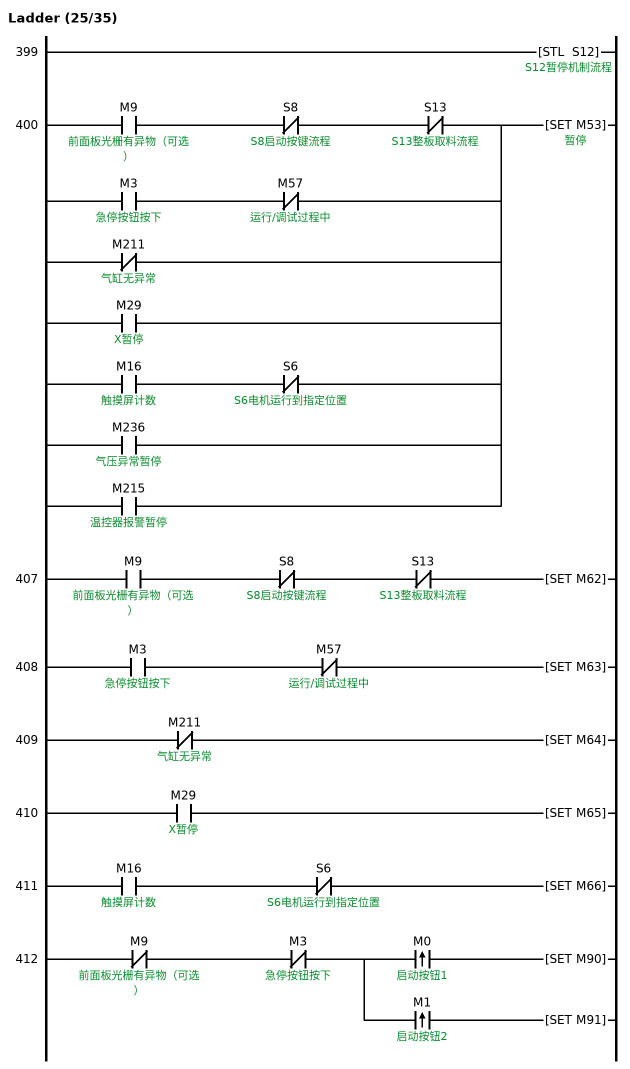
[picture p24: Ladder rows 399-412]
STL    S12	; S12暂停机制流程
LD     M9	; 前面板光栅有异物（可选）
ANI    S8	; S8启动按键流程
ANI    S13	; S13整板取料流程
LD     M3	; 急停按钮按下
ANI    M57	; 运行/调试过程中
ORB
ORI    M211	; 气缸无异常
OR     M29	; X暂停
LD     M16	; 触摸屏计数
ANI    S6	; S6电机运行到指定位置
ORB
OR     M236	; 气压异常暂停
OR     M215	; 温控器报警暂停
SET    M53	; 暂停
LD     M9	; 前面板光栅有异物（可选）
ANI    S8	; S8启动按键流程
ANI    S13	; S13整板取料流程
SET    M62
LD     M3	; 急停按钮按下
ANI    M57	; 运行/调试过程中
SET    M63
LDI    M211	; 气缸无异常
SET    M64
LD     M29	; X暂停
SET    M65
LD     M16	; 触摸屏计数
ANI    S6	; S6电机运行到指定位置
SET    M66
LDI    M9	; 前面板光栅有异物（可选）
ANI    M3	; 急停按钮按下
MPS
ANDP   M0	; 启动按钮1
SET    M90
MPP
ANDP   M1	; 启动按钮2
SET    M91

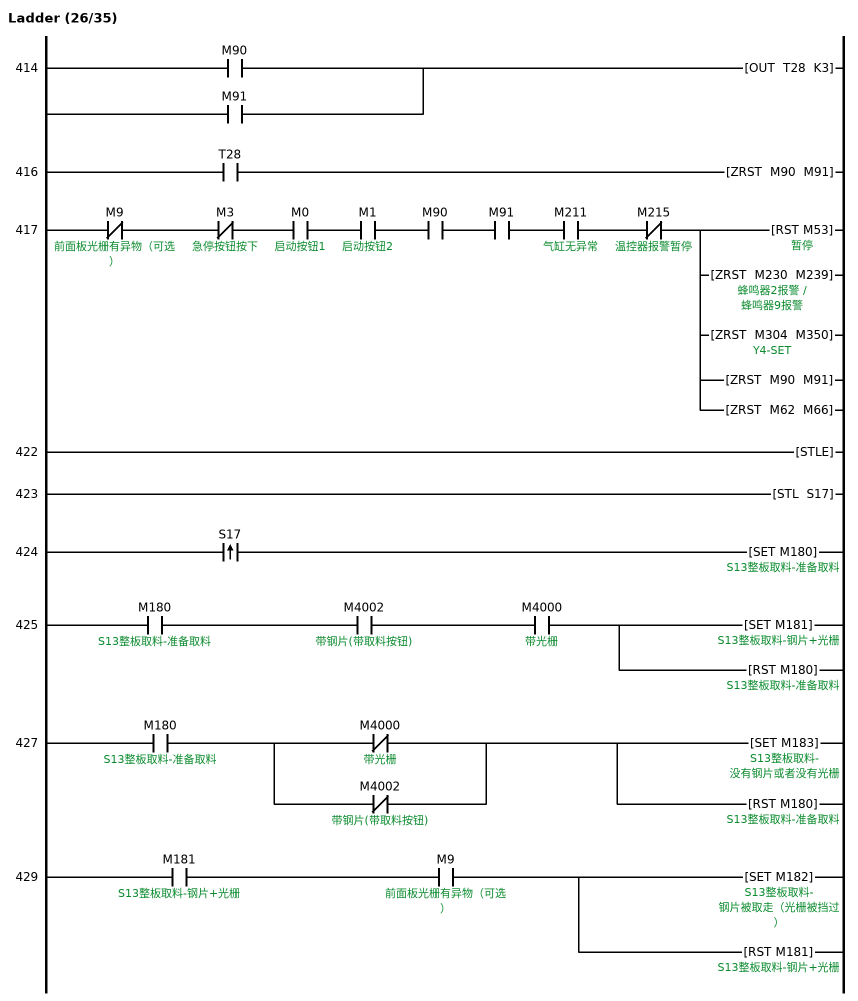
LD     M90
OR     M91
OUT    T28 K3
LD     T28
ZRST   M90 M91
LDI    M9	; 前面板光栅有异物（可选）
ANI    M3	; 急停按钮按下
AND    M0	; 启动按钮1
AND    M1	; 启动按钮2
AND    M90
AND    M91
AND    M211	; 气缸无异常
ANI    M215	; 温控器报警暂停
RST    M53	; 暂停
ZRST   M230 M239	; 蜂鸣器2报警 / 蜂鸣器9报警
ZRST   M304 M350	; Y4-SET
ZRST   M90 M91
ZRST   M62 M66
STLE
STL    S17
LDP    S17
SET    M180	; S13整板取料-准备取料
LD     M180	; S13整板取料-准备取料
AND    M4002	; 带钢片(带取料按钮)
AND    M4000	; 带光栅
SET    M181	; S13整板取料-钢片+光栅
RST    M180	; S13整板取料-准备取料
LD     M180	; S13整板取料-准备取料
LDI    M4000	; 带光栅
ORI    M4002	; 带钢片(带取料按钮)
ANB
SET    M183	; S13整板取料-没有钢片或者没有光栅
RST    M180	; S13整板取料-准备取料
LD     M181	; S13整板取料-钢片+光栅
AND    M9	; 前面板光栅有异物（可选）
SET    M182	; S13整板取料-钢片被取走（光栅被挡过）
RST    M181	; S13整板取料-钢片+光栅

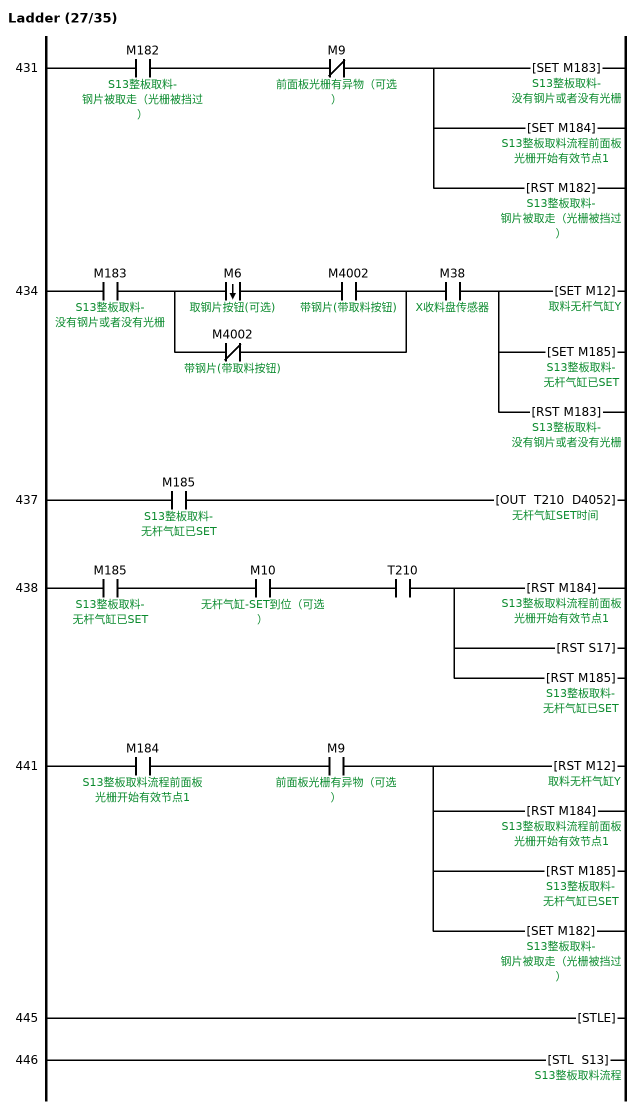
LD     M182	; S13整板取料-钢片被取走（光栅被挡过）
ANI    M9	; 前面板光栅有异物（可选）
SET    M183	; S13整板取料-没有钢片或者没有光栅
SET    M184	; S13整板取料流程前面板光栅开始有效节点1
RST    M182	; S13整板取料-钢片被取走（光栅被挡过）
LD     M183	; S13整板取料-没有钢片或者没有光栅
LDF    M6	; 取钢片按钮(可选)
AND    M4002	; 带钢片(带取料按钮)
ORI    M4002	; 带钢片(带取料按钮)
ANB
AND    M38	; X收料盘传感器
SET    M12	; 取料无杆气缸Y
SET    M185	; S13整板取料-无杆气缸已SET
RST    M183	; S13整板取料-没有钢片或者没有光栅
LD     M185	; S13整板取料-无杆气缸已SET
OUT    T210 D4052	; 无杆气缸SET时间
LD     M185	; S13整板取料-无杆气缸已SET
AND    M10	; 无杆气缸-SET到位（可选）
AND    T210
RST    M184	; S13整板取料流程前面板光栅开始有效节点1
RST    S17
RST    M185	; S13整板取料-无杆气缸已SET
LD     M184	; S13整板取料流程前面板光栅开始有效节点1
AND    M9	; 前面板光栅有异物（可选）
RST    M12	; 取料无杆气缸Y
RST    M184	; S13整板取料流程前面板光栅开始有效节点1
RST    M185	; S13整板取料-无杆气缸已SET
SET    M182	; S13整板取料-钢片被取走（光栅被挡过）
STLE
STL    S13	; S13整板取料流程

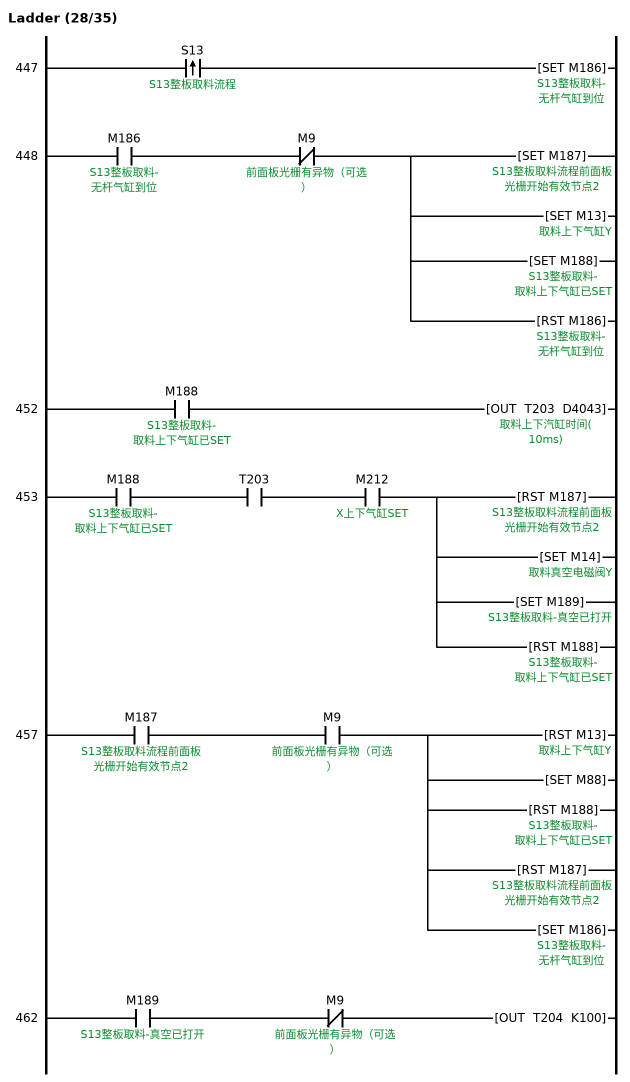
LDP    S13	; S13整板取料流程
SET    M186	; S13整板取料-无杆气缸到位
LD     M186	; S13整板取料-无杆气缸到位
ANI    M9	; 前面板光栅有异物（可选）
SET    M187	; S13整板取料流程前面板光栅开始有效节点2
SET    M13	; 取料上下气缸Y
SET    M188	; S13整板取料-取料上下气缸已SET
RST    M186	; S13整板取料-无杆气缸到位
LD     M188	; S13整板取料-取料上下气缸已SET
OUT    T203 D4043	; 取料上下汽缸时间(10ms)
LD     M188	; S13整板取料-取料上下气缸已SET
AND    T203
AND    M212	; X上下气缸SET
RST    M187	; S13整板取料流程前面板光栅开始有效节点2
SET    M14	; 取料真空电磁阀Y
SET    M189	; S13整板取料-真空已打开
RST    M188	; S13整板取料-取料上下气缸已SET
LD     M187	; S13整板取料流程前面板光栅开始有效节点2
AND    M9	; 前面板光栅有异物（可选）
RST    M13	; 取料上下气缸Y
SET    M88
RST    M188	; S13整板取料-取料上下气缸已SET
RST    M187	; S13整板取料流程前面板光栅开始有效节点2
SET    M186	; S13整板取料-无杆气缸到位
LD     M189	; S13整板取料-真空已打开
ANI    M9	; 前面板光栅有异物（可选）
OUT    T204 K100

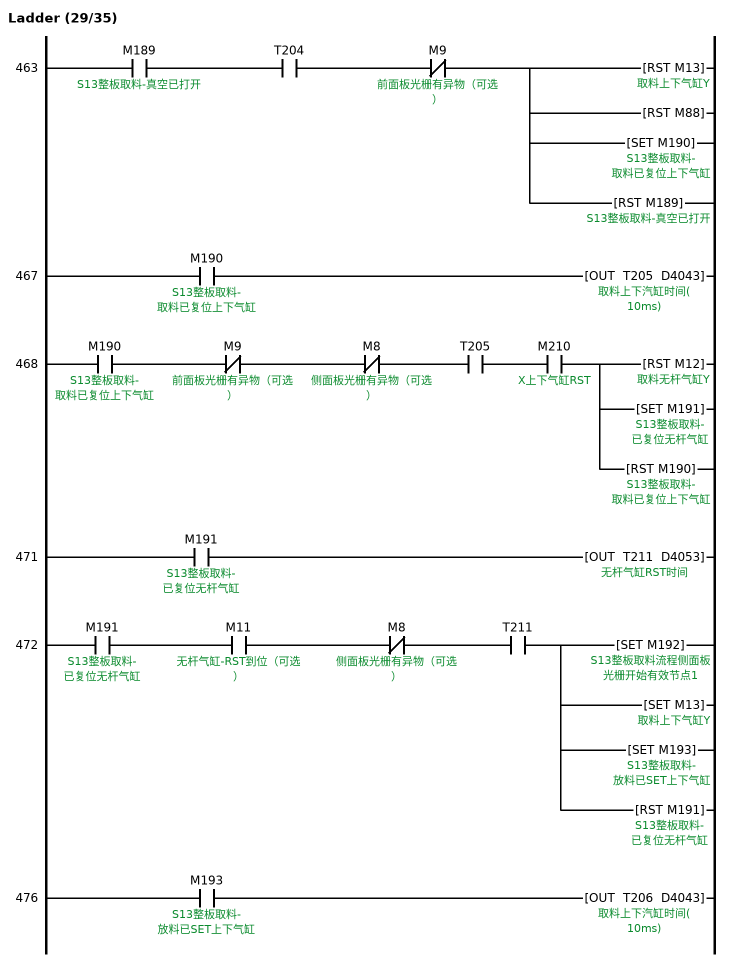
LD     M189	; S13整板取料-真空已打开
AND    T204
ANI    M9	; 前面板光栅有异物（可选）
RST    M13	; 取料上下气缸Y
RST    M88
SET    M190	; S13整板取料-取料已复位上下气缸
RST    M189	; S13整板取料-真空已打开
LD     M190	; S13整板取料-取料已复位上下气缸
OUT    T205 D4043	; 取料上下汽缸时间(10ms)
LD     M190	; S13整板取料-取料已复位上下气缸
ANI    M9	; 前面板光栅有异物（可选）
ANI    M8	; 侧面板光栅有异物（可选）
AND    T205
AND    M210	; X上下气缸RST
RST    M12	; 取料无杆气缸Y
SET    M191	; S13整板取料-已复位无杆气缸
RST    M190	; S13整板取料-取料已复位上下气缸
LD     M191	; S13整板取料-已复位无杆气缸
OUT    T211 D4053	; 无杆气缸RST时间
LD     M191	; S13整板取料-已复位无杆气缸
AND    M11	; 无杆气缸-RST到位（可选）
ANI    M8	; 侧面板光栅有异物（可选）
AND    T211
SET    M192	; S13整板取料流程侧面板光栅开始有效节点1
SET    M13	; 取料上下气缸Y
SET    M193	; S13整板取料-放料已SET上下气缸
RST    M191	; S13整板取料-已复位无杆气缸
LD     M193	; S13整板取料-放料已SET上下气缸
OUT    T206 D4043	; 取料上下汽缸时间(10ms)

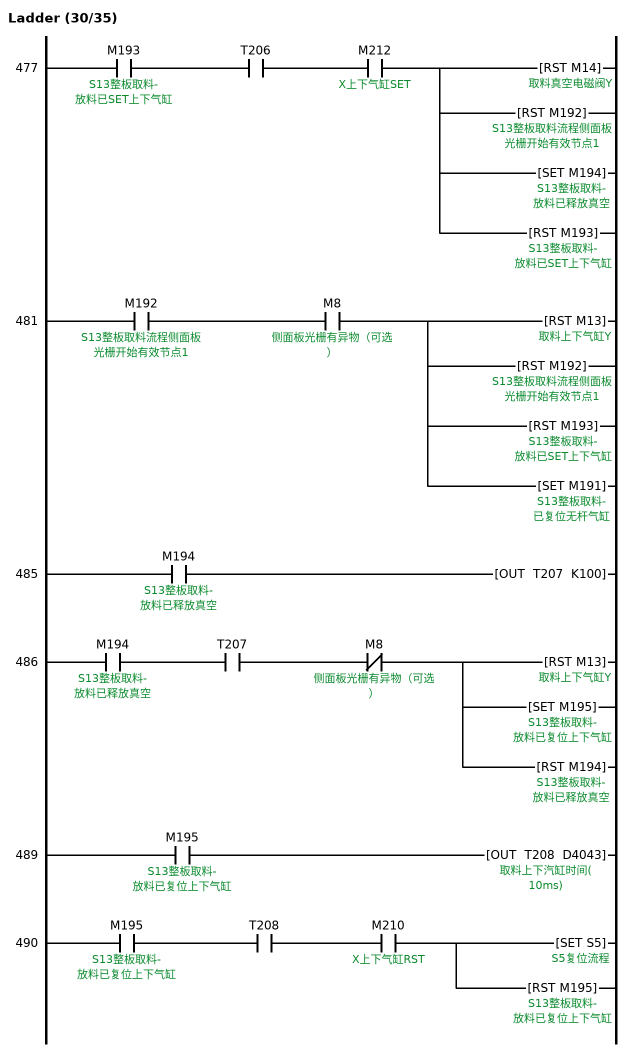
LD     M193	; S13整板取料-放料已SET上下气缸
AND    T206
AND    M212	; X上下气缸SET
RST    M14	; 取料真空电磁阀Y
RST    M192	; S13整板取料流程侧面板光栅开始有效节点1
SET    M194	; S13整板取料-放料已释放真空
RST    M193	; S13整板取料-放料已SET上下气缸
LD     M192	; S13整板取料流程侧面板光栅开始有效节点1
AND    M8	; 侧面板光栅有异物（可选）
RST    M13	; 取料上下气缸Y
RST    M192	; S13整板取料流程侧面板光栅开始有效节点1
RST    M193	; S13整板取料-放料已SET上下气缸
SET    M191	; S13整板取料-已复位无杆气缸
LD     M194	; S13整板取料-放料已释放真空
OUT    T207 K100
LD     M194	; S13整板取料-放料已释放真空
AND    T207
ANI    M8	; 侧面板光栅有异物（可选）
RST    M13	; 取料上下气缸Y
SET    M195	; S13整板取料-放料已复位上下气缸
RST    M194	; S13整板取料-放料已释放真空
LD     M195	; S13整板取料-放料已复位上下气缸
OUT    T208 D4043	; 取料上下汽缸时间(10ms)
LD     M195	; S13整板取料-放料已复位上下气缸
AND    T208
AND    M210	; X上下气缸RST
SET    S5	; S5复位流程
RST    M195	; S13整板取料-放料已复位上下气缸

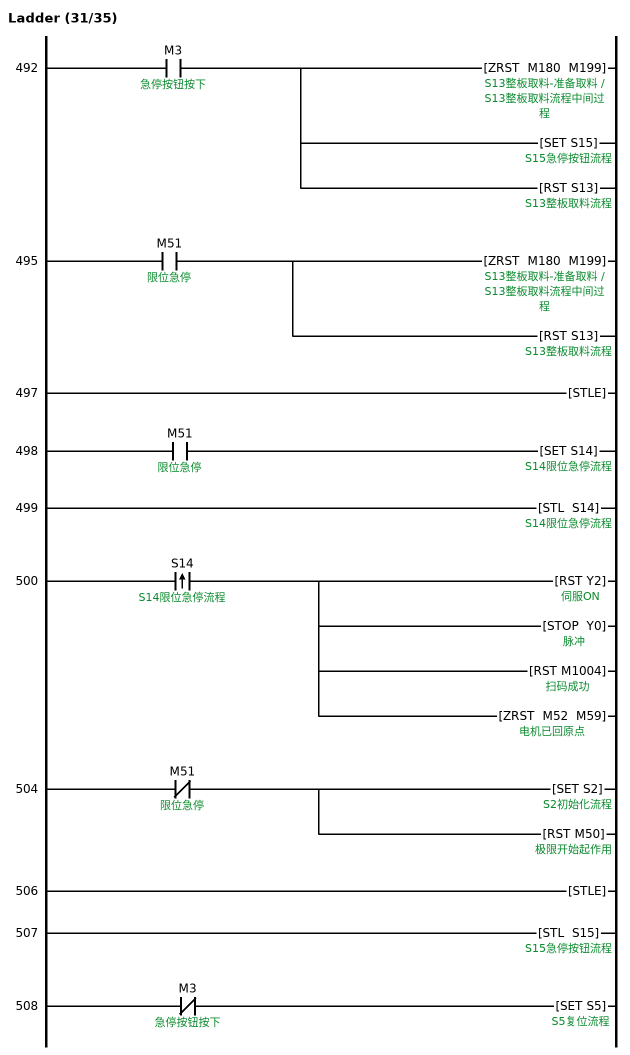
LD     M3	; 急停按钮按下
ZRST   M180 M199	; S13整板取料-准备取料 / S13整板取料流程中间过程
SET    S15	; S15急停按钮流程
RST    S13	; S13整板取料流程
LD     M51	; 限位急停
ZRST   M180 M199	; S13整板取料-准备取料 / S13整板取料流程中间过程
RST    S13	; S13整板取料流程
STLE
LD     M51	; 限位急停
SET    S14	; S14限位急停流程
STL    S14	; S14限位急停流程
LDP    S14	; S14限位急停流程
RST    Y2	; 伺服ON
STOP   Y0	; 脉冲
RST    M1004	; 扫码成功
ZRST   M52 M59	; 电机已回原点
LDI    M51	; 限位急停
SET    S2	; S2初始化流程
RST    M50	; 极限开始起作用
STLE
STL    S15	; S15急停按钮流程
LDI    M3	; 急停按钮按下
SET    S5	; S5复位流程

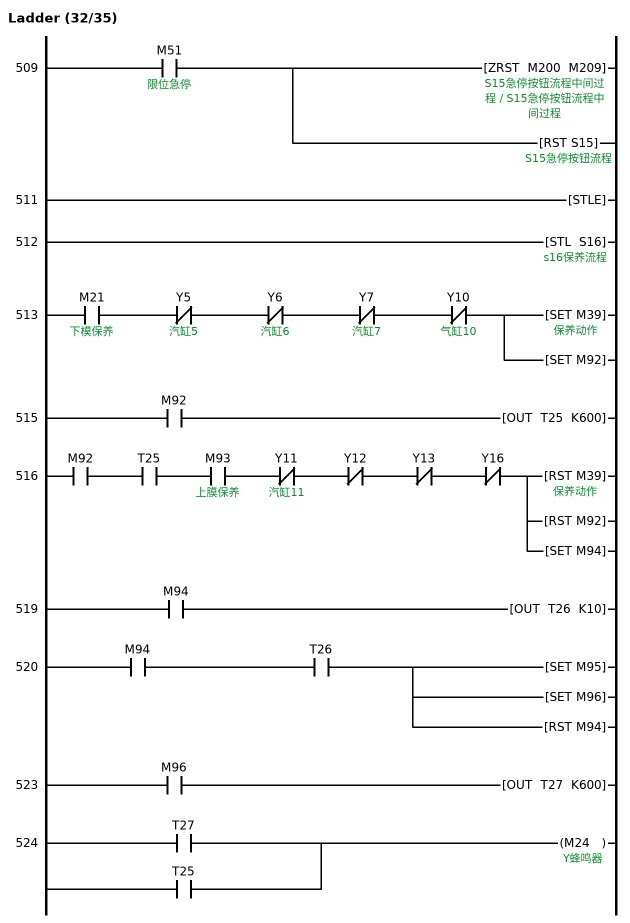
LD     M51	; 限位急停
ZRST   M200 M209	; S15急停按钮流程中间过程 / S15急停按钮流程中间过程
RST    S15	; S15急停按钮流程
STLE
STL    S16	; s16保养流程
LD     M21	; 下模保养
ANI    Y5	; 汽缸5
ANI    Y6	; 汽缸6
ANI    Y7	; 汽缸7
ANI    Y10	; 气缸10
SET    M39	; 保养动作
SET    M92
LD     M92
OUT    T25 K600
LD     M92
AND    T25
AND    M93	; 上膜保养
ANI    Y11	; 汽缸11
ANI    Y12
ANI    Y13
ANI    Y16
RST    M39	; 保养动作
RST    M92
SET    M94
LD     M94
OUT    T26 K10
LD     M94
AND    T26
SET    M95
SET    M96
RST    M94
LD     M96
OUT    T27 K600
LD     T27
OR     T25
OUT    M24	; Y蜂鸣器

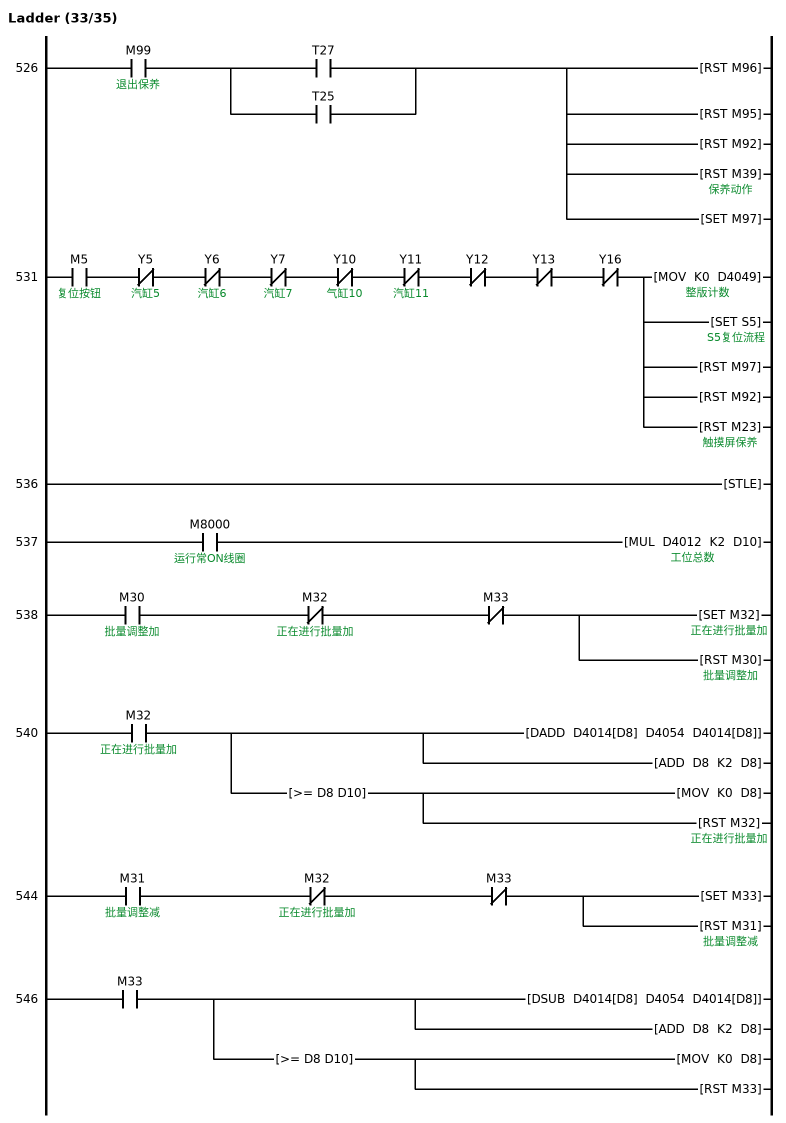
LD     M99	; 退出保养
LD     T27
OR     T25
ANB
RST    M96
RST    M95
RST    M92
RST    M39	; 保养动作
SET    M97
LD     M5	; 复位按钮
ANI    Y5	; 汽缸5
ANI    Y6	; 汽缸6
ANI    Y7	; 汽缸7
ANI    Y10	; 气缸10
ANI    Y11	; 汽缸11
ANI    Y12
ANI    Y13
ANI    Y16
MOV    K0 D4049	; 整版计数
SET    S5	; S5复位流程
RST    M97
RST    M92
RST    M23	; 触摸屏保养
STLE
LD     M8000	; 运行常ON线圈
MUL    D4012 K2 D10	; 工位总数
LD     M30	; 批量调整加
ANI    M32	; 正在进行批量加
ANI    M33
SET    M32	; 正在进行批量加
RST    M30	; 批量调整加
LD     M32	; 正在进行批量加
DADD   D4014[D8] D4054 D4014[D8]
ADD    D8 K2 D8
AND>=  D8 D10
MOV    K0 D8
RST    M32	; 正在进行批量加
LD     M31	; 批量调整减
ANI    M32	; 正在进行批量加
ANI    M33
SET    M33
RST    M31	; 批量调整减
LD     M33
DSUB   D4014[D8] D4054 D4014[D8]
ADD    D8 K2 D8
AND>=  D8 D10
MOV    K0 D8
RST    M33

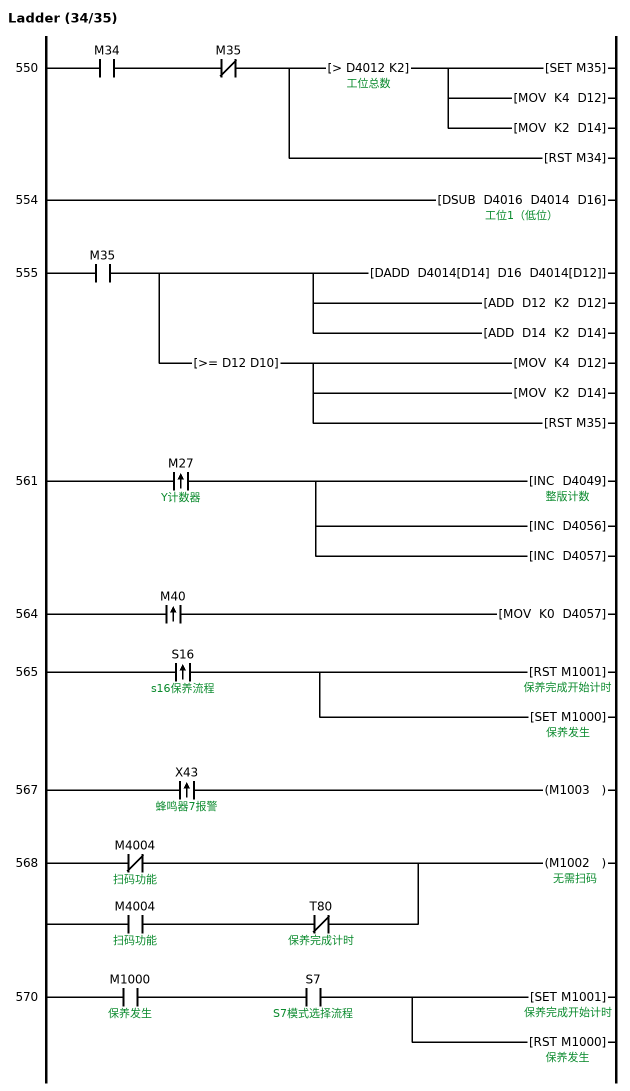
LD     M34
ANI    M35
MPS
AND>   D4012 K2	; 工位总数
SET    M35
MOV    K4 D12
MOV    K2 D14
MPP
RST    M34
DSUB   D4016 D4014 D16	; 工位1（低位）
LD     M35
DADD   D4014[D14] D16 D4014[D12]
ADD    D12 K2 D12
ADD    D14 K2 D14
AND>=  D12 D10
MOV    K4 D12
MOV    K2 D14
RST    M35
LDP    M27	; Y计数器
INC    D4049	; 整版计数
INC    D4056
INC    D4057
LDP    M40
MOV    K0 D4057
LDP    S16	; s16保养流程
RST    M1001	; 保养完成开始计时
SET    M1000	; 保养发生
LDP    X43	; 蜂鸣器7报警
OUT    M1003
LDI    M4004	; 扫码功能
LD     M4004	; 扫码功能
ANI    T80	; 保养完成计时
ORB
OUT    M1002	; 无需扫码
LD     M1000	; 保养发生
AND    S7	; S7模式选择流程
SET    M1001	; 保养完成开始计时
RST    M1000	; 保养发生

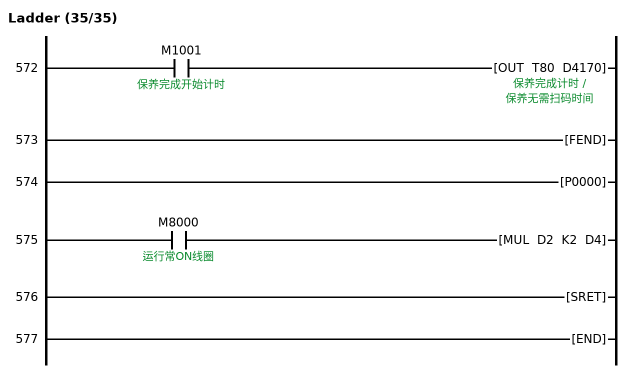
LD     M1001	; 保养完成开始计时
OUT    T80 D4170	; 保养完成计时 / 保养无需扫码时间
FEND
P0000
LD     M8000	; 运行常ON线圈
MUL    D2 K2 D4
SRET
END

COMMENTS (devices not used above)
X10	Y4-RST
X44	蜂鸣器8报警
X100	Y10-SET-2
X101	Y11-SET-1
X102	Y11-SET-2
X103	Y12-SET-1
X104	Y12-SET-2
X105	Y13-SET-1
X106	Y13-SET-2
X107	Y14-SET
M19	换行
M60	保养中间过程
M61	保养中间过程
M103	S2初始化流程中间过程
M104	S2初始化流程中间过程
M105	S2初始化流程中间过程
M106	S2初始化流程中间过程
M107	S2初始化流程中间过程
M108	S2初始化流程中间过程
M112	S4回原点流程中间过程
M116	S4回原点流程中间过程
M117	S4回原点流程中间过程
M118	S4回原点流程中间过程
M121	S6电机运行到指定位置中间过程
M122	S6电机运行到指定位置中间过程
M123	S6电机运行到指定位置中间过程
M124	S6电机运行到指定位置中间过程
M125	S6电机运行到指定位置中间过程
M126	S6电机运行到指定位置中间过程
M127	S6电机运行到指定位置中间过程
M128	S6电机运行到指定位置中间过程
M136	S5复位流程中间过程
M137	S5复位流程中间过程
M138	S5复位流程中间过程
M143	S7模式选择流程中间过程
M144	S7模式选择流程中间过程
M145	S7模式选择流程中间过程
M146	S7模式选择流程中间过程
M147	S7模式选择流程中间过程
M148	S7模式选择流程中间过程
M154	S8启动按键流程中间过程
M155	S8启动按键流程中间过程
M156	S8启动按键流程中间过程
M157	S8启动按键流程中间过程
M158	S8启动按键流程中间过程
M165	S9运行流程中间过程
M166	S9运行流程中间过程
M167	S9运行流程中间过程
M168	S9运行流程中间过程
M174	S10调试模式中间过程
M175	S10调试模式中间过程
M176	S10调试模式中间过程
M177	S10调试模式中间过程
M178	S10调试模式中间过程
M196	S13整板取料流程中间过程
M197	S13整板取料流程前面板光栅开始有效节点2
M198	S13整板取料流程中间过程
M201	S15急停按钮流程中间过程
M202	S15急停按钮流程中间过程
M203	S15急停按钮流程中间过程
M204	S15急停按钮流程中间过程
M205	S15急停按钮流程中间过程
M206	S15急停按钮流程中间过程
M207	S15急停按钮流程中间过程
M208	S15急停按钮流程中间过程
M303	Y3置位异常
M323	Y3复位异常
M324	Y4-RST
S104	S104 R Y6 Y7 Y10 
S105	S105 R Y4
S106	S106 R Y14
S107	S107 S Y14
S108	S108 R Y5 Y10
S109	S109 R Y3
S110	S110 S Y6
S111	S111 S Y16
S112	S112 S Y12
S113	S113 R Y12 Y16
S114	S114 S Y11
S115	S115 R Y11
S116	S116 S 14
S117	S117 R 14
T40	注意此处修改
T45	注意此处修改
T404	Y4-SET
T414	Y11置位异常
T454	Y4-RST
T464	Y11复位异常
D5004	注意此处修改
D5010	Y4压合时间
D5012	Y5压合时间
D5014	Y6压合时间
D5016	Y7压合时间
D5018	Y10压合时间